INTERFACE I_Quaternion


METHOD GetNorm : LREAL
END_METHOD


METHOD GetNormSq : LREAL
END_METHOD


METHOD ToString : T_MaxString
END_METHOD


PROPERTY w : LREAL
GET
END_GET
END_PROPERTY


PROPERTY x : LREAL
GET
END_GET
END_PROPERTY


PROPERTY y : LREAL
GET
END_GET
END_PROPERTY


PROPERTY z : LREAL
GET
END_GET
END_PROPERTY

END_INTERFACE

(* stored: Version 1.1.0.1
   Itf I_Quaternion: Id {d6831b85-2c4c-4d0a-b783-213a1dbe68b8}
   Method GetNorm: Id {2ff59caa-1a8e-4d8e-8340-5d7de889d133}
   Method GetNormSq: Id {1105fc22-644a-4770-a3b5-b7cc0d09cdd0}
   Method ToString: Id {b259c3aa-8217-4bd1-aeee-d6eb659fa7d1}
   Property w: Id {1e2facaf-ec30-4cec-90d5-e084127bc0f9}
   Get Get: Id {8f4d5b69-a2e5-49ed-8aef-4c45ad79831d}
   Property x: Id {56eeaf1d-5bbb-48cf-8238-3c241aab42ea}
   Get Get: Id {a553d82c-7968-4025-a8a0-75a845fd2364}
   Property y: Id {3c928912-1d5a-4787-b094-1d4c4d3f69a6}
   Get Get: Id {8460eb31-b5ae-4d41-a2fd-301f1d48fa0c}
   Property z: Id {79d3f71a-6337-44c6-b3ca-3387c045552b}
   Get Get: Id {9239d992-e814-4b2c-ab53-fcb33ccb1074} *)
